(* IEC 61131-3 sources: plcc/crates/plcc-codegen/src/compiler, 2 files *)

(* ---- real_string.st ---- *)
(* SPDX-License-Identifier: MPL-2.0 *)
(* REAL/LREAL <-> STRING, compiled into a module only when it uses them
   (see compiler/ondemand.rs). *)

FUNCTION __PLCC_FLOAT_TO_STRING : STRING
VAR_INPUT
    X : LREAL;
    DIGITS : INT;   (* significant digits: 7 for REAL, 15 for LREAL *)
END_VAR
VAR
    ax : LREAL;
    e : DINT;
    m : LINT;
    lim : LINT;
    ds : STRING;
    nd : INT;
    k : INT;
    s : STRING;
    ex : DINT;
END_VAR
IF X <> X THEN
    __PLCC_FLOAT_TO_STRING := 'NaN';
    RETURN;
END_IF;
ax := ABS(X);
IF ax > LREAL#1.7976931348623157E308 THEN
    IF X < 0.0 THEN
        __PLCC_FLOAT_TO_STRING := '-INF';
    ELSE
        __PLCC_FLOAT_TO_STRING := 'INF';
    END_IF;
    RETURN;
END_IF;
IF ax = 0.0 THEN
    __PLCC_FLOAT_TO_STRING := '0';
    RETURN;
END_IF;
(* ax = m * 10^(e - DIGITS + 1), with m holding exactly DIGITS digits. *)
e := TRUNC(FLOOR(LOG(ax)));
m := LREAL_TO_LINT(ax * EXPT(LREAL#10.0, DIGITS - 1 - e));
lim := LREAL_TO_LINT(EXPT(LREAL#10.0, DIGITS));
IF m >= lim THEN
    m := m / 10;
    e := e + 1;
ELSIF m < lim / 10 THEN
    m := m * 10;
    e := e - 1;
END_IF;
ds := LINT_TO_STRING(m);
(* Significant digits without trailing zeros. *)
nd := DIGITS;
WHILE nd > 1 AND MID(ds, 1, nd) = '0' DO
    nd := nd - 1;
END_WHILE;
IF X < 0.0 THEN
    s := '-';
END_IF;
IF e >= -5 AND e < DIGITS THEN
    IF e >= 0 THEN
        (* Integer part: the first e+1 digits, padded with zeros. *)
        FOR k := 1 TO DINT_TO_INT(e) + 1 DO
            IF k <= nd THEN
                s := CONCAT(s, MID(ds, 1, k));
            ELSE
                s := CONCAT(s, '0');
            END_IF;
        END_FOR;
        IF nd > e + 1 THEN
            s := CONCAT(s, '.');
            s := CONCAT(s, MID(ds, nd - DINT_TO_INT(e) - 1, DINT_TO_INT(e) + 2));
        END_IF;
    ELSE
        s := CONCAT(s, '0.');
        FOR k := 1 TO DINT_TO_INT(-e) - 1 DO
            s := CONCAT(s, '0');
        END_FOR;
        s := CONCAT(s, LEFT(ds, nd));
    END_IF;
ELSE
    s := CONCAT(s, LEFT(ds, 1));
    IF nd > 1 THEN
        s := CONCAT(s, '.');
        s := CONCAT(s, MID(ds, nd - 1, 2));
    END_IF;
    IF e < 0 THEN
        s := CONCAT(s, 'E-');
        ex := -e;
    ELSE
        s := CONCAT(s, 'E+');
        ex := e;
    END_IF;
    IF ex < 10 THEN
        s := CONCAT(s, '0');
    END_IF;
    s := CONCAT(s, DINT_TO_STRING(ex));
END_IF;
__PLCC_FLOAT_TO_STRING := s;
END_FUNCTION

FUNCTION REAL_TO_STRING : STRING
VAR_INPUT X : REAL; END_VAR
REAL_TO_STRING := __PLCC_FLOAT_TO_STRING(REAL_TO_LREAL(X), 7);
END_FUNCTION

FUNCTION LREAL_TO_STRING : STRING
VAR_INPUT X : LREAL; END_VAR
LREAL_TO_STRING := __PLCC_FLOAT_TO_STRING(X, 15);
END_FUNCTION

FUNCTION STRING_TO_LREAL : LREAL
VAR_INPUT S : STRING; END_VAR
VAR
    pt : POINTER TO BYTE;
    v : LREAL;
    neg : BOOL;
    scale : DINT;
    e : DINT;
    eneg : BOOL;
END_VAR
pt := ADR(S);
WHILE pt^ = 32 DO
    pt := pt + 1;
END_WHILE;
IF pt^ = 45 THEN
    neg := TRUE;
    pt := pt + 1;
ELSIF pt^ = 43 THEN
    pt := pt + 1;
END_IF;
WHILE pt^ >= 48 AND pt^ <= 57 DO
    v := v * 10.0 + BYTE_TO_LREAL(pt^ - 48);
    pt := pt + 1;
END_WHILE;
IF pt^ = 46 THEN
    pt := pt + 1;
    WHILE pt^ >= 48 AND pt^ <= 57 DO
        v := v * 10.0 + BYTE_TO_LREAL(pt^ - 48);
        scale := scale - 1;
        pt := pt + 1;
    END_WHILE;
END_IF;
IF pt^ = 69 OR pt^ = 101 THEN
    pt := pt + 1;
    IF pt^ = 45 THEN
        eneg := TRUE;
        pt := pt + 1;
    ELSIF pt^ = 43 THEN
        pt := pt + 1;
    END_IF;
    WHILE pt^ >= 48 AND pt^ <= 57 DO
        e := e * 10 + BYTE_TO_DINT(pt^ - 48);
        pt := pt + 1;
    END_WHILE;
    IF eneg THEN
        e := -e;
    END_IF;
END_IF;
scale := scale + e;
IF scale <> 0 THEN
    v := v * EXPT(LREAL#10.0, scale);
END_IF;
IF neg THEN
    v := -v;
END_IF;
STRING_TO_LREAL := v;
END_FUNCTION

FUNCTION STRING_TO_REAL : REAL
VAR_INPUT S : STRING; END_VAR
STRING_TO_REAL := LREAL_TO_REAL(STRING_TO_LREAL(S));
END_FUNCTION

(* ---- time_string.st ---- *)
(* SPDX-License-Identifier: MPL-2.0 *)
(* TIME / date values -> STRING, in the literal syntax CODESYS prints, compiled
   into a module only when it uses them (see compiler/ondemand.rs). Date and
   time-of-day fields are not zero-padded, as in the CODESYS help's examples:
   DATE_TO_STRING(D#1970-1-1) = 'D#1970-1-1', TOD_TO_STRING(TOD#12:0:1) =
   'TOD#12:0:1'; milliseconds are always three digits ('TOD#2:3:4.005'). *)

(* 'T#1d2h3m4s5ms', units that are 0 left out; 'T#0ms' for zero. With NS,
   sub-millisecond units (us, ns) are printed too (LTIME). *)
FUNCTION __PLCC_DURATION_TO_STRING : STRING
VAR_INPUT
    NSV : LINT;
    PREFIX : STRING;
    NS : BOOL;
END_VAR
VAR
    v : LINT;
    s : STRING;
    part : LINT;
END_VAR
s := PREFIX;
v := NSV;
IF v < 0 THEN
    s := CONCAT(s, '-');
    v := -v;
END_IF;
IF NOT NS THEN
    v := v / 1000000;   (* whole milliseconds *)
    IF v = 0 THEN
        __PLCC_DURATION_TO_STRING := CONCAT(s, '0ms');
        RETURN;
    END_IF;
    part := v / 86400000; IF part > 0 THEN s := CONCAT(s, CONCAT(LINT_TO_STRING(part), 'd')); END_IF;
    part := (v / 3600000) MOD 24; IF part > 0 THEN s := CONCAT(s, CONCAT(LINT_TO_STRING(part), 'h')); END_IF;
    part := (v / 60000) MOD 60; IF part > 0 THEN s := CONCAT(s, CONCAT(LINT_TO_STRING(part), 'm')); END_IF;
    part := (v / 1000) MOD 60; IF part > 0 THEN s := CONCAT(s, CONCAT(LINT_TO_STRING(part), 's')); END_IF;
    part := v MOD 1000; IF part > 0 THEN s := CONCAT(s, CONCAT(LINT_TO_STRING(part), 'ms')); END_IF;
ELSE
    IF v = 0 THEN
        __PLCC_DURATION_TO_STRING := CONCAT(s, '0ns');
        RETURN;
    END_IF;
    part := v / 86400000000000; IF part > 0 THEN s := CONCAT(s, CONCAT(LINT_TO_STRING(part), 'd')); END_IF;
    part := (v / 3600000000000) MOD 24; IF part > 0 THEN s := CONCAT(s, CONCAT(LINT_TO_STRING(part), 'h')); END_IF;
    part := (v / 60000000000) MOD 60; IF part > 0 THEN s := CONCAT(s, CONCAT(LINT_TO_STRING(part), 'm')); END_IF;
    part := (v / 1000000000) MOD 60; IF part > 0 THEN s := CONCAT(s, CONCAT(LINT_TO_STRING(part), 's')); END_IF;
    part := (v / 1000000) MOD 1000; IF part > 0 THEN s := CONCAT(s, CONCAT(LINT_TO_STRING(part), 'ms')); END_IF;
    part := (v / 1000) MOD 1000; IF part > 0 THEN s := CONCAT(s, CONCAT(LINT_TO_STRING(part), 'us')); END_IF;
    part := v MOD 1000; IF part > 0 THEN s := CONCAT(s, CONCAT(LINT_TO_STRING(part), 'ns')); END_IF;
END_IF;
__PLCC_DURATION_TO_STRING := s;
END_FUNCTION

(* 'YYYY-MM-DD' of nanoseconds since 1970-01-01 (Howard Hinnant's
   civil_from_days). *)
FUNCTION __PLCC_DATE_PART : STRING
VAR_INPUT NSV : LINT; END_VAR
VAR z : LINT; era : LINT; doe : LINT; yoe : LINT; y : LINT; doy : LINT; mp : LINT; d : LINT; m : LINT; END_VAR
z := NSV / 86400000000000;
IF NSV < 0 AND NSV MOD 86400000000000 <> 0 THEN z := z - 1; END_IF;
z := z + 719468;
IF z >= 0 THEN era := z / 146097; ELSE era := (z - 146096) / 146097; END_IF;
doe := z - era * 146097;
yoe := (doe - doe / 1460 + doe / 36524 - doe / 146096) / 365;
y := yoe + era * 400;
doy := doe - (365 * yoe + yoe / 4 - yoe / 100);
mp := (5 * doy + 2) / 153;
d := doy - (153 * mp + 2) / 5 + 1;
IF mp < 10 THEN m := mp + 3; ELSE m := mp - 9; END_IF;
IF m <= 2 THEN y := y + 1; END_IF;
__PLCC_DATE_PART := CONCAT(CONCAT(CONCAT(LINT_TO_STRING(y), '-'), CONCAT(LINT_TO_STRING(m), '-')), LINT_TO_STRING(d));
END_FUNCTION

(* 'h:m:s' plus '.mmm' when there are milliseconds. *)
FUNCTION __PLCC_TOD_PART : STRING
VAR_INPUT NSV : LINT; END_VAR
VAR t : LINT; s : STRING; ms : LINT; END_VAR
t := NSV MOD 86400000000000;
IF t < 0 THEN t := t + 86400000000000; END_IF;
t := t / 1000000;
s := CONCAT(CONCAT(LINT_TO_STRING(t / 3600000), ':'), CONCAT(LINT_TO_STRING(t / 60000 MOD 60), ':'));
s := CONCAT(s, LINT_TO_STRING(t / 1000 MOD 60));
ms := t MOD 1000;
IF ms > 0 THEN
    IF ms < 10 THEN
        s := CONCAT(s, '.00');
    ELSIF ms < 100 THEN
        s := CONCAT(s, '.0');
    ELSE
        s := CONCAT(s, '.');
    END_IF;
    s := CONCAT(s, LINT_TO_STRING(ms));
END_IF;
__PLCC_TOD_PART := s;
END_FUNCTION

FUNCTION TIME_TO_STRING : STRING
VAR_INPUT X : TIME; END_VAR
TIME_TO_STRING := __PLCC_DURATION_TO_STRING(LTIME_TO_LINT(TIME_TO_LTIME(X)), 'T#', FALSE);
END_FUNCTION

FUNCTION LTIME_TO_STRING : STRING
VAR_INPUT X : LTIME; END_VAR
LTIME_TO_STRING := __PLCC_DURATION_TO_STRING(LTIME_TO_LINT(X), 'LTIME#', TRUE);
END_FUNCTION

FUNCTION DATE_TO_STRING : STRING
VAR_INPUT X : DATE; END_VAR
DATE_TO_STRING := CONCAT('D#', __PLCC_DATE_PART(LDATE_TO_LINT(DATE_TO_LDATE(X))));
END_FUNCTION

FUNCTION TOD_TO_STRING : STRING
VAR_INPUT X : TOD; END_VAR
TOD_TO_STRING := CONCAT('TOD#', __PLCC_TOD_PART(LTOD_TO_LINT(TOD_TO_LTOD(X))));
END_FUNCTION

FUNCTION DT_TO_STRING : STRING
VAR_INPUT X : DT; END_VAR
VAR n : LINT; END_VAR
n := LDT_TO_LINT(DT_TO_LDT(X));
DT_TO_STRING := CONCAT(CONCAT(CONCAT('DT#', __PLCC_DATE_PART(n)), '-'), __PLCC_TOD_PART(n));
END_FUNCTION
